Staubli VAL3: TrajPallet.dtx

public TrajPointItem tData
  [0]
    TrajectoryItem tSuper
      [0]
        num distance
        num moveType
        num nTime
        num nStop
        num nTcpAction
        string comment
        bool toStop
        mdesc nom_speed = {vel=450, tmax=600, rmax=9999, leave=30, reach=30}
        InstrItem iInstr[3]
          [0]
            string sType
            string sData
          [1]
            string sType
            string sData
          [2]
            string sType
            string sData
        num nMoveId
    pointRx pPoint = {fatherId=fFrame[0]}
    num nType
public frame fFrame = {fatherId=fReference[0]}
public num nIndexTool
public string sID
public trsf trAppro[2]
public trsf trDepart[2]
public num nX = 1
public num nY = 1
public num nZ = 1
public num nIndex
public num nDistanceXYZ[3]
  [0] = 1
  [1] = 1
  [2] = 1
public string sAction
public pointRx pO = {fatherId=fReference[0]}
public pointRx pX = {fatherId=fReference[0]}
public pointRx pY = {fatherId=fReference[0]}
public pointRx pZ = {fatherId=fReference[0]}
public num nSpeedApproach = 500
public num nSpeedDepart = 500
public num nIndexFrame
public frame fReference = {fatherId=world[0]}
